(* PLC project Tc2_Utilities.INSERT2 Demo, tc3-libraries-kb TwinCAT 3.1 *)
(* stored: creationDateTime 2026-05-10T16:00:00, modificationDateTime 2026-05-10T16:00:00 *)

PROGRAM P_Demo_INSERT2
  VAR
    rResult : BOOL;  (* INSERT2 返回值 *)
    bRun : BOOL;  (* 触发一次调用 *)
    sIn : STRING(255) := 'foobar';  (* 测试用本地变量 *)
    sIns : STRING(31) := 'XYZ';  (* 测试用本地变量 *)
    sOut : STRING(255);  (* 测试用本地变量 *)
  END_VAR

            // ============================================================
// Tc2_Utilities.INSERT2 演示程序（FUNCTION）
// ============================================================
// 验证步骤：
//   1. 引用 Tc2_Utilities
//   2. 编译 + 登录
//   3. 强制 bRun := TRUE 一个周期
//   4. 在线监视 rResult / 各 demo 变量
// ============================================================

IF bRun THEN
    rResult := INSERT2(ADR(sIn), ADR(sIns), ADR(sOut), SIZEOF(sOut), 3);
    bRun := FALSE;
END_IF;

          
END_PROGRAM
